TYPE ST_EP9224_SlaveIn :
STRUCT
	nOutput	:ARRAY [1..EP9224_NUM_CHANNELS] OF BYTE;
END_STRUCT
END_TYPE

(* stored: Version 1.1.0.1, ProductVersion 3.1.4024.9
   DUT ST_EP9224_SlaveIn: Id {52f2e45d-1c4e-4ba4-9ee8-9840493eb27d} *)
